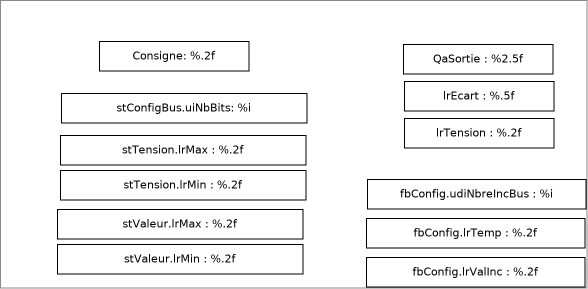
VISUALIZATION vi_ConvertAnalog_1  // 588x289
    Rectangle (99,41 150x30), "Consigne: %.2f", text variable: fbConvertTachoToNumSpeed.IaEntree
        OnMouseDown: write the text variable via Default
    Rectangle (61,93 246x30), "stConfigBus.uiNbBits: %i", text variable: fbConvertTachoToNumSpeed.fbConfig.uiNbreBitBus
        OnMouseDown: write the text variable via Default
    Rectangle (60,135 246x30), "stTension.lrMax : %.2f", text variable: fbConvertTachoToNumSpeed.fbConfig.stTension.lrMax
        OnMouseDown: write the text variable via Default
    Rectangle (60,170 246x30), "stTension.lrMin : %.2f", text variable: fbConvertTachoToNumSpeed.fbConfig.stTension.lrMin
        OnMouseDown: write the text variable via Default
    Rectangle (57,209 246x30), "stValeur.lrMax : %.2f", text variable: fbConvertTachoToNumSpeed.fbConfig.stValeur.lrMax
        OnMouseDown: write the text variable via Default
    Rectangle (57,244 246x30), "stValeur.lrMin : %.2f", text variable: fbConvertTachoToNumSpeed.fbConfig.stValeur.lrMin
        OnMouseDown: write the text variable via Default
    Rectangle (403,44 150x30), "QaSortie : %2.5f", text variable: fbConvertTachoToNumSpeed.lrValeur
    Rectangle (367,179 219x30), "fbConfig.udiNbreIncBus : %i", text variable: fbConvertTachoToNumSpeed.fbConfig.udiNbreIncBus
    Rectangle (366,218 219x30), "fbConfig.lrTemp : %.2f", text variable: fbConvertTachoToNumSpeed.fbConfig.lrTemp
    Rectangle (404,81 150x30), "lrEcart : %.5f", text variable: fbConvertTachoToNumSpeed.lrEcart
    Rectangle (404,118 150x30), "lrTension : %.2f", text variable: fbConvertTachoToNumSpeed.lrTension
    Rectangle (366,257 219x30), "fbConfig.lrValInc : %.2f", text variable: fbConvertTachoToNumSpeed.fbConfig.lrValInc
END_VISUALIZATION

(* stored: Version 1.1.0.1, ProductVersion 3.1.4020.6
   Visu vi_ConvertAnalog_1: Id {11c2e472-76cc-4006-a22a-c3ca69361ca4} *)
